// LS Electric XG5000 project: 0122 PLC 데이터 계산기
// PLC LSPLC

PROGRAM NewProgram (task: 스캔 프로그램)

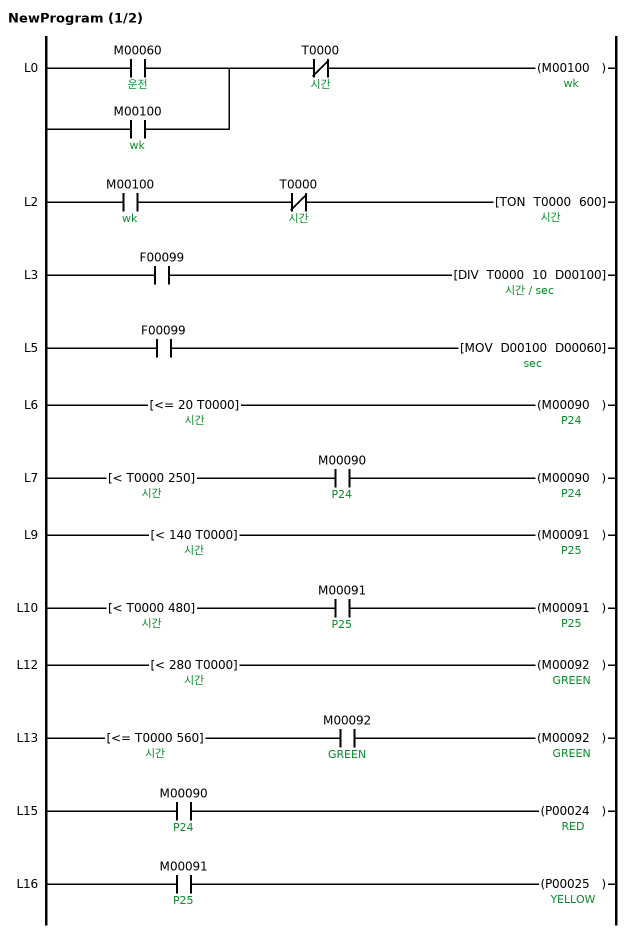
; L0
LOAD      M00060	// 운전
OR        M00100	// wk
AND NOT   T0000	// 시간
OUT       M00100	// wk
; L2
LOAD      M00100	// wk
AND NOT   T0000	// 시간
TON       T0000 600	// 시간
; L3
LOAD      F00099
DIV       T0000 10 D00100	// 시간 / sec
; L5
LOAD      F00099
MOV       D00100 D00060	// sec
; L6
LOAD<=    20 T0000	// 시간
OUT       M00090	// P24
; L7
LOAD<     T0000 250	// 시간
AND       M00090	// P24
OUT       M00090	// P24
; L9
LOAD<     140 T0000	// 시간
OUT       M00091	// P25
; L10
LOAD<     T0000 480	// 시간
AND       M00091	// P25
OUT       M00091	// P25
; L12
LOAD<     280 T0000	// 시간
OUT       M00092	// GREEN
; L13
LOAD<=    T0000 560	// 시간
AND       M00092	// GREEN
OUT       M00092	// GREEN
; L15
LOAD      M00090	// P24
OUT       P00024	// RED
; L16
LOAD      M00091	// P25
OUT       P00025	// YELLOW

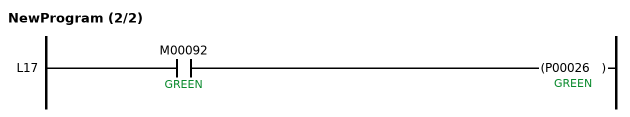
; L17
LOAD      M00092	// GREEN
OUT       P00026	// GREEN

VARIABLES AND COMMENTS (devices not used above)
M00010	BIT	스위치 1
D00000	WORD	전번
M00001	BIT	스위치2
D00022	WORD	현재카운터수
M00002	BIT	스위치3
M00003	BIT	카운터
M00004	BIT	카운터 리셋
C0000	BIT/WORD	카운트
M00000	BIT	스위치1
M00041	BIT	더하기
D00030	WORD	입력1
D00032	WORD	입력2
D00040	WORD	결과
M00042	BIT	빼기
M00043	BIT	곱하기
M00044	BIT	나누기
M00045	BIT	CLR